FUNCTION_BLOCK Payload_A IMPLEMENTS I_Payload_A
VAR_INPUT
END_VAR
VAR_OUTPUT
END_VAR
VAR
	nPayload : INT;
END_VAR

END_FUNCTION_BLOCK

(* stored: Version 1.1.0.1, ProductVersion 3.1.4024.2
   POU Payload_A: Id {68e569a0-88d4-46f8-9a9e-3121423266f2}, SpecialFunc None *)
